// LS Electric XG5000 project: PMixer
// PLC LSPLC

PROGRAM NewProgram (task: 스캔 프로그램)

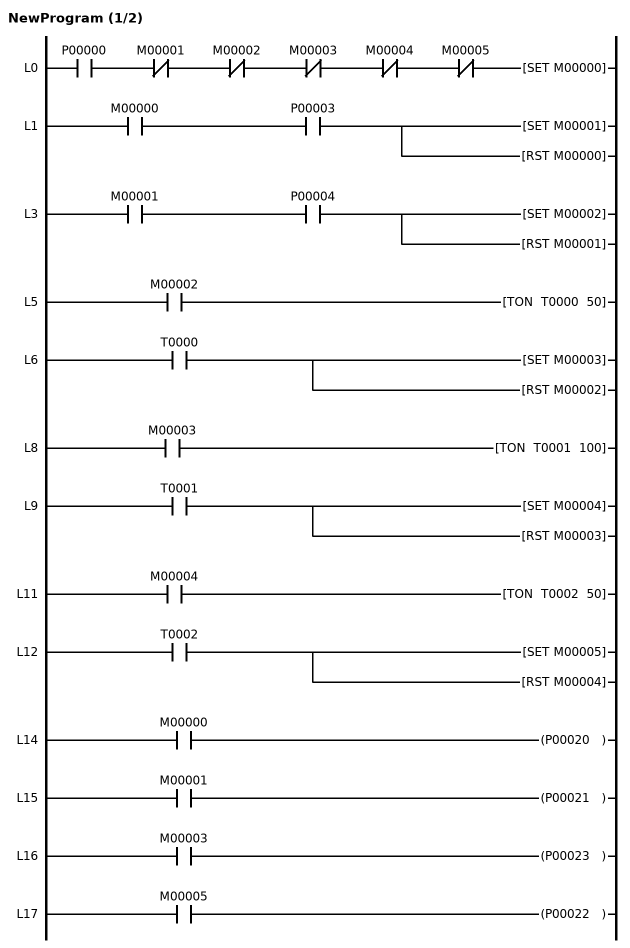
; L0
LOAD      P00000
AND NOT   M00001
AND NOT   M00002
AND NOT   M00003
AND NOT   M00004
AND NOT   M00005
SET       M00000
; L1
LOAD      M00000
AND       P00003
SET       M00001
RST       M00000
; L3
LOAD      M00001
AND       P00004
SET       M00002
RST       M00001
; L5
LOAD      M00002
TON       T0000 50
; L6
LOAD      T0000
SET       M00003
RST       M00002
; L8
LOAD      M00003
TON       T0001 100
; L9
LOAD      T0001
SET       M00004
RST       M00003
; L11
LOAD      M00004
TON       T0002 50
; L12
LOAD      T0002
SET       M00005
RST       M00004
; L14
LOAD      M00000
OUT       P00020
; L15
LOAD      M00001
OUT       P00021
; L16
LOAD      M00003
OUT       P00023
; L17
LOAD      M00005
OUT       P00022

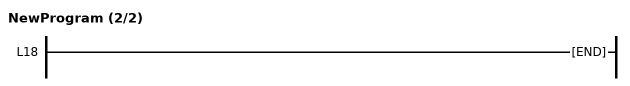
; L18
END